FUNCTION_BLOCK FB_AxisBase
VAR_INPUT
	bPowerEnable 	: BOOL := TRUE;
	bPosEnable		: BOOL := TRUE;
	bNegEnable		: BOOL := TRUE;
	bStop			: BOOL;
	bReset 			: BOOL;
	fOverride		: LREAL := 100.0;
END_VAR
VAR_OUTPUT
	bAxisRdy		: BOOL;
	bError			: BOOL;
	nErrId			: UDINT;
END_VAR
VAR
	m_axis		: AXIS_REF;	

	m_fb_power 	: MC_Power;
	m_fb_reset	: MC_Reset;
	m_fb_stop  	: MC_Stop;
	m_fb_state	: MC_ReadStatus;

	m_axis_status 	: ST_AxisStatus;
	m_state			: ST_McOutputs;
	st_fbMcStopOut	: ST_McOutputs;
	
END_VAR

m_fb_state(Axis:= m_axis, Enable:= TRUE);


m_fb_power(
	Axis 				:= m_axis,
	Enable 				:= bPowerEnable,
	Override 			:= fOverride,
	Enable_Positive 	:= bPosEnable,
	Enable_Negative 	:= bNegEnable,
);
	
m_fb_reset(
	Axis := m_axis,
	Execute := bReset
	);

	
m_fb_stop(
	Axis := m_axis,
	Execute := bStop,
	);


bStop 	:= FALSE;
bReset 	:= FALSE;

bAxisRdy	:= m_fb_power.Status;
bError 		:= m_fb_power.Error 		OR m_fb_reset.Error		OR m_fb_stop.Error OR m_fb_state.Error;
nErrId 		:= m_fb_power.ErrorID OR m_fb_reset.ErrorID	OR m_fb_stop.ErrorID OR m_fb_state.ErrorID;

END_FUNCTION_BLOCK

(* stored: Version 1.1.0.1, ProductVersion 3.1.4024.13
   POU FB_AxisBase: Id {53216d91-db3c-4d91-ac3f-174d20d70566}, SpecialFunc None *)
